(*
    This testsuite runs two tests. One that is enabled (and that is supposed to fail), and one that is disabled (and
    even though it also is failing is not supposed to run).
*)
{attribute 'call_after_init'}
FUNCTION_BLOCK FB_CreateDisabledTest EXTENDS TcUnit.FB_TestSuite IMPLEMENTS TcUnit.I_RunnableTestSuite
VAR
    Assert : TcUnit.FB_Assert;
END_VAR

METHOD FB_init : BOOL
VAR_INPUT
	bInitRetains : BOOL; // if TRUE, the retain variables are initialized (warm start / cold start)
	bInCopyCode : BOOL;  // if TRUE, the instance afterwards gets moved into the copy code (online change)
END_VAR
SUPER^.RegisterTestSuite(THIS^);
END_METHOD

METHOD RunTests : TCUNIT.E_TestSuiteRunState
TestEnabled();
TestDisabled();

RunTests := TCUNIT.E_TestSuiteRunState.FINISHED;
END_METHOD

METHOD PRIVATE TestDisabled
VAR
    a : BOOL := FALSE;
    b : BOOL := TRUE;
END_VAR
TEST('DISABLED_ThisShouldNotExecute');

Assert.AssertEquals(Expected := a,
                    Actual := b,
                    Message := 'A does not equal B');
END_METHOD

METHOD PRIVATE TestEnabled
VAR
    a : BOOL := TRUE;
    b : BOOL := FALSE;
END_VAR
TEST('TestEnabled');

Assert.AssertEquals(Expected := a,
                    Actual := b,
                    Message := 'A does not equal B');
END_METHOD

END_FUNCTION_BLOCK

(* stored: Version 1.1.0.1, ProductVersion 3.1.4022.16
   POU FB_CreateDisabledTest: Id {3f1093ff-32d2-455a-8cf0-190014c55a4c}, SpecialFunc None
   Method FB_init: Id {301e9f58-092a-49ca-8343-33e6bc16c7de}
   Method RunTests: Id {c91bd153-d1fb-4a6a-8ec2-77d6ab3f7087}
   Method TestDisabled: Id {773db475-8255-416d-8669-8526d3357b4d}
   Method TestEnabled: Id {aaa74956-ecdb-40ff-a4da-e0ad237c9503} *)
